// TIA Portal V17 export
// export: Created 2026-04-13T11:12:45.4428722Z, ExportSetting WithDefaults, DisplayName Totally Integrated Automation Portal, DisplayVersion V17 Update 4, DisplayName TIA Portal Openness, DisplayVersion V17 Update 4, DisplayName TIA Portal Version Control Interface, DisplayVersion V17, DisplayName SINAMICS Startdrive Advanced, DisplayVersion V17, DisplayName SINAMICS Startdrive G130, G150, S120, S150, SINAMICS MV, S210, DisplayVersion V17, DisplayName SINAMICS Startdrive G110M, G120, G120C, G120D, G120P, G115D, DisplayVersion V17, DisplayName STEP 7 Professional, DisplayVersion V17 Update 4, DisplayName STEP 7 Safety, DisplayVersion V17, DisplayName WinCC Professional, DisplayVersion V17 Update 4
VAR_GLOBAL   // PLC tag table "M"
   MMC脉冲反吹 AT %M400.0 : Bool;
   MJF进温自整定 AT %M400.1 : Bool;
   MSF送风机 AT %M400.2 : Bool;
   MSF送风机风扇 AT %M400.3 : Bool;
   MDJ电加热器 AT %M400.4 : Bool;
   MLX离心雾化 AT %M400.5 : Bool;
   MLX离心雾化风扇 AT %M400.6 : Bool;
   MLX离心雾化油泵 AT %M400.7 : Bool;
   MJL进料泵 AT %M401.0 : Bool;
   MJL进料泵风扇 AT %M401.1 : Bool;
   MYF引风机 AT %M401.2 : Bool;
   MYF引风机风扇 AT %M401.3 : Bool;
   MSF输送风机 AT %M401.4 : Bool;
   MSF输送加热器 AT %M401.5 : Bool;
   MRJ溶剂排液泵 AT %M401.6 : Bool;
   MCC除尘脉冲 AT %M401.7 : Bool;
   MFM蜂鸣器 AT %M402.0 : Bool;
   MZS指示灯 AT %M402.1 : Bool;
   MYS钥匙开关 AT %M402.2 : Bool;
   MQX清洗溶剂罐进氮阀 AT %M402.3 : Bool;
   MBD补氮阀 AT %M402.4 : Bool;
   MJD进氮阀 AT %M402.5 : Bool;
   MJF进风蒸汽开关阀 AT %M402.6 : Bool;
   MJF进风蒸汽比例调节阀 AT %M402.7 : Bool;
   MJF进风蒸汽排水阀 AT %M403.0 : Bool;
   MQX清洗溶剂进阀 AT %M403.1 : Bool;
   MQX清洗溶剂出阀 AT %M403.2 : Bool;
   MWL物料进阀 AT %M403.3 : Bool;
   MYJ一级出料上阀 AT %M403.4 : Bool;
   MYJ一级出料下阀 AT %M403.5 : Bool;
   MEJ二级出料上阀 AT %M403.6 : Bool;
   MEJ二级出料下阀 AT %M403.7 : Bool;
   MCC除尘出料上阀 AT %M404.0 : Bool;
   MCC除尘出料下阀 AT %M404.1 : Bool;
   MKS开式排风隔断阀 AT %M404.2 : Bool;
   MBS闭式排风隔断阀 AT %M404.3 : Bool;
   MKS开式进风隔断阀 AT %M404.4 : Bool;
   MBS闭式进风隔断阀 AT %M404.5 : Bool;
   MYJ一级冷却水阀 AT %M404.6 : Bool;
   MYJ二级冷冻水阀 AT %M404.7 : Bool;
   MYJ一级排液阀 AT %M405.0 : Bool;
   MEJ二级排液阀 AT %M405.1 : Bool;
   MCW除雾排液阀 AT %M405.2 : Bool;
   MRJ溶剂回收排放阀 AT %M405.3 : Bool;
   MHF回风蒸汽开关阀 AT %M405.4 : Bool;
   MHF回风蒸汽调节阀 AT %M405.5 : Bool;
   MHF回风蒸汽排水阀 AT %M405.6 : Bool;
   MXY泄压阀 AT %M405.7 : Bool;
   MPH平衡比例调节阀 AT %M406.0 : Bool;
   MJF进风冷却水阀 AT %M406.1 : Bool;
   MSS输送进风阀 AT %M406.2 : Bool;
   MSS输送出料上阀 AT %M406.3 : Bool;
   MSS输送出料下阀 AT %M406.4 : Bool;
   MQL气流雾化阀 AT %M406.5 : Bool;
   MZT主塔气锤 AT %M406.6 : Bool;
   MYJ一级旋风气锤 AT %M406.7 : Bool;
   MYJ一级缓存振荡器 AT %M407.0 : Bool;
   MEJ二级旋风气锤 AT %M407.1 : Bool;
   MEJ二级缓存震荡器 AT %M407.2 : Bool;
   MCC除尘气锤 AT %M407.3 : Bool;
   MCC除尘缓存震荡器 AT %M407.4 : Bool;
   MTD塔顶清洗球阀 AT %M407.5 : Bool;
   MQG气缸升降阀 AT %M407.6 : Bool;
   MZT主塔清洗进水阀 AT %M407.7 : Bool;
   MXF旋风管道清洗阀 AT %M408.0 : Bool;
   MYJ一级旋风清洗阀 AT %M408.1 : Bool;
   MEJ二级旋风清洗阀 AT %M408.2 : Bool;
   MCC除尘管道清洗阀 AT %M408.3 : Bool;
   MCC除尘清洗阀 AT %M408.4 : Bool;
   MSS输送管路清洗阀 AT %M408.5 : Bool;
   MLC料仓清洗阀 AT %M408.6 : Bool;
   MJR加热清洗阀 AT %M408.7 : Bool;
   MWK蜗壳清洗阀 AT %M409.0 : Bool;
   MCF出风高效清洗阀 AT %M409.1 : Bool;
   MZT主塔排水阀 AT %M409.2 : Bool;
   MSS输送管路排水阀 AT %M409.3 : Bool;
   MLC料仓清洗排水阀 AT %M409.4 : Bool;
   MSF送风机清洗阀 AT %M409.5 : Bool;
   MYF引风机清洗阀 AT %M409.6 : Bool;
   MYJ一级冷凝清洗阀 AT %M409.7 : Bool;
   MEJ二级冷凝清洗阀 AT %M410.0 : Bool;
   MSF送风机排水阀 AT %M410.1 : Bool;
   MYF引风机排水阀 AT %M410.2 : Bool;
   MEJ二级冷冻水阀 AT %M410.3 : Bool;
   MQX清洗伸缩气缸 AT %M410.4 : Bool;
   MFK放空比例调节阀 AT %M410.5 : Bool;
   MHF回风加热比例调节阀 AT %M410.6 : Bool;
   MJF进风加热比例调节阀 AT %M410.7 : Bool;
   MYJ一级出料 AT %M411.0 : Bool;
   MEJ二级出料 AT %M411.1 : Bool;
   MBD布袋出料 AT %M411.2 : Bool;
   MSS输送出料 AT %M411.3 : Bool;
   MQG气缸升 AT %M411.4 : Bool;
   MQG气缸降 AT %M411.5 : Bool;
   MYH氧含仪隔断阀 AT %M411.6 : Bool;
   MSN室内排水隔膜泵 AT %M412.0 : Bool;
   MSS输送自整定 AT %M412.1 : Bool;
   MSS输送加热 AT %M412.2 : Bool;
   MBY100 AT %M412.3 : Bool;
   MBY101 AT %M412.4 : Bool;
   MAS室外回水阀 AT %M412.5 : Bool;
   MAS室内回水阀 AT %M412.6 : Bool;
   MSN室内清洗总阀 AT %M412.7 : Bool;
   MHS回水隔断阀1 AT %M413.0 : Bool;
   MAB进水隔断阀 AT %M413.1 : Bool;
   MHSQ回水隔断阀1 AT %M413.2 : Bool;
   MABQ进水隔断阀 AT %M413.3 : Bool;
   MLG料罐清洗阀 AT %M413.4 : Bool;
   MHF回风温度加热 AT %M413.5 : Bool;
   MHF回风加热自整定 AT %M413.6 : Bool;
   MSC四参数控制 AT %M413.7 : Bool;
   MMC脉冲周期_PID AT %M414.0 : Bool;
   MMC脉冲周期_进料 AT %M414.1 : Bool;
   MLS料水手动调节 AT %M414.2 : Bool;
   MXT心跳接受信号 AT %M414.3 : Bool;
   MCS纯水洗请求 AT %M414.4 : Bool;
   MJS碱水洗请求 AT %M414.5 : Bool;
   MRJ溶剂请求 AT %M414.6 : Bool;
   MYG压干请求 AT %M414.7 : Bool;
   MQR确认 AT %M415.0 : Bool;
   MSC四参数手动调节 AT %M415.1 : Bool;
   MZT暂停辅助 AT %M415.2 : Bool;
   MSC四参数开辅助 AT %M415.3 : Bool;
   MSC四参数关辅助 AT %M415.4 : Bool;
   MJL进料调节 AT %M415.5 : Bool;
   MSC四参数调节 AT %M415.6 : Bool;
   MSC四参数手动状态 AT %M415.7 : Bool;
   MJL进料手动状态 AT %M416.1 : Bool;
   MSS输送系统 AT %M416.2 : Bool;
   MJS进水调节 AT %M416.3 : Bool;
   MLS料水系统调节 AT %M416.4 : Bool;
   MKS开始清洗 AT %M416.5 : Bool;
   MJS结束清洗 AT %M416.6 : Bool;
   MZB准备清洗 AT %M416.7 : Bool;
   MCZ初状态 AT %M417.0 : Bool;
   MZD自动清洗 AT %M417.1 : Bool;
   MSD手动_纯水清洗 AT %M417.2 : Bool;
   MSD手动_碱水清洗 AT %M417.3 : Bool;
   MQX清洗辅助 AT %M417.4 : Bool;
   "MSD手动_溶剂清洗(1)" AT %M417.5 : Bool;
   MSD手动_溶剂清洗 AT %M417.6 : Bool;
   MZT主塔伸缩气缸 AT %M417.7 : Bool;
   MZT主塔清洗 AT %M418.0 : Bool;
   MZT总通路 AT %M418.1 : Bool;
   MXY泄压请求 AT %M418.2 : Bool;
   QXY泄压请求 AT %M418.3 : Bool;
   MBJ本机调试模式 AT %M418.4 : Bool;
   MSD手动_二纯水清洗 AT %M418.5 : Bool;
   MFZ仿真调试 AT %M418.6 : Bool;
   MSB设备振打 AT %M418.7 : Bool;
   MQZ前置水阀 AT %M419.0 : Bool;
   MYJ一级旋风振打锤 AT %M419.1 : Bool;
   MEJ二级旋风振打锤 AT %M419.2 : Bool;
   MYJ一级旋风振荡器 AT %M419.3 : Bool;
   MAQ安全停机 AT %M419.4 : Bool;
   MZS注射水请求 AT %M419.5 : Bool;
   MSJ水进程泵 AT %M419.6 : Bool;
   MRJ溶剂进程泵 AT %M419.7 : Bool;
   MGS供水泵 AT %M420.0 : Bool;
   MRC热纯自动洗 AT %M420.1 : Bool;
   MRC热纯加热 AT %M420.2 : Bool;
   MBD本地调试 AT %M420.3 : Bool;
   MRS热水洗请求 AT %M420.4 : Bool;
   MGD管道压力手动调节 AT %M420.5 : Bool;
   MPS排水运行标志 AT %M420.6 : Bool;
END_VAR
